// TIA Portal project "Lan-mahai birakaria" (V15.1)

(* hardware
DEVICE "S7-1200 station_1"  S7-1200 Station
   slot 0: "Rack_0"  S7-1200 Rack  Rack  V1.0
   slot 1: "PLC_1"  CPU 1214C AC/DC/Rly  6ES7 214-1BG40-0XB0  V4.0
*)

// ===== PLC "PLC_1"  CPU 1214C AC/DC/Rly =====

VAR_GLOBAL   // PLC tag table "Tabla de variables estándar"
   "Etapa 0" AT %M0.0 : Bool;
   "Etapa 1" AT %M0.1 : Bool;
   "Etapa 2" AT %M0.2 : Bool;
   "Etapa 11" AT %M0.4 : Bool;
   "Etapa 12" AT %M0.5 : Bool;
   "Etapa 20" AT %M0.6 : Bool;
   "Etapa 21" AT %M0.7 : Bool;
   "Etapa 22" AT %M1.0 : Bool;
   "Etapa 23" AT %M1.1 : Bool;
   "Etapa 24" AT %M1.2 : Bool;
   "Etapa 30" AT %M1.3 : Bool;
   "Etapa 31" AT %M1.4 : Bool;
   "Etapa 32" AT %M1.5 : Bool;
   "Etapa 33" AT %M1.6 : Bool;
   "Etapa 34" AT %M1.7 : Bool;
   "Etapa 35" AT %M2.0 : Bool;
   "Etapa 10" AT %M0.3 : Bool;
   "M" AT %I0.0 : Bool;
   "A" AT %I0.1 : Bool;
   "DI0" AT %I0.2 : Bool;
   "DI1" AT %I0.3 : Bool;
   "DI2" AT %I0.4 : Bool;
   "TA" AT %I0.5 : Bool;
   "TB" AT %I0.6 : Bool;
   "TTA" AT %I0.7 : Bool;
   "TTB" AT %I1.0 : Bool;
   "C1R" AT %I1.1 : Bool;
   "C1F" AT %I1.2 : Bool;
   "C2R" AT %I1.3 : Bool;
   "C2F" AT %I1.4 : Bool;
   "S1" AT %Q0.0 : Bool;
   "S2" AT %Q0.1 : Bool;
   "R1" AT %Q0.2 : Bool;
   "R2" AT %Q0.3 : Bool;
   "C1" AT %Q0.4 : Bool;
   "C2" AT %Q0.5 : Bool;
   "MT" AT %Q0.6 : Bool;
   "MP" AT %Q0.7 : Bool;
   "PE" AT %I1.5 : Bool;
END_VAR

// folder: System blocks/Program resources

DATA_BLOCK "Temporizador 1"   // DB1
{ S7_Optimized_Access := 'TRUE' }
AUTHOR : Simatic
FAMILY : IEC
NAME : IEC_TMR
VERSION : 1.0
// stored: InstanceOfName IEC_TIMER
"IEC_TIMER"
BEGIN
END_DATA_BLOCK

DATA_BLOCK "Temporizador 2"   // DB4
{ S7_Optimized_Access := 'TRUE' }
AUTHOR : Simatic
FAMILY : IEC
NAME : IEC_TMR
VERSION : 1.0
// stored: InstanceOfName IEC_TIMER
"IEC_TIMER"
BEGIN
END_DATA_BLOCK

// folder: (top level)

ORGANIZATION_BLOCK "Main"   // OB1, LAD, ProgramCycle
TITLE = "Main Program Sweep (Cycle)"
{ S7_Optimized_Access := 'TRUE' }
VERSION : 0.1
   VAR_INPUT
      Initial_Call : Bool;   // Initial call of this OB
      Remanence : Bool;   // =True, if remanent data are available
   END_VAR
BEGIN

REGION Network 1
   // Etapa 1
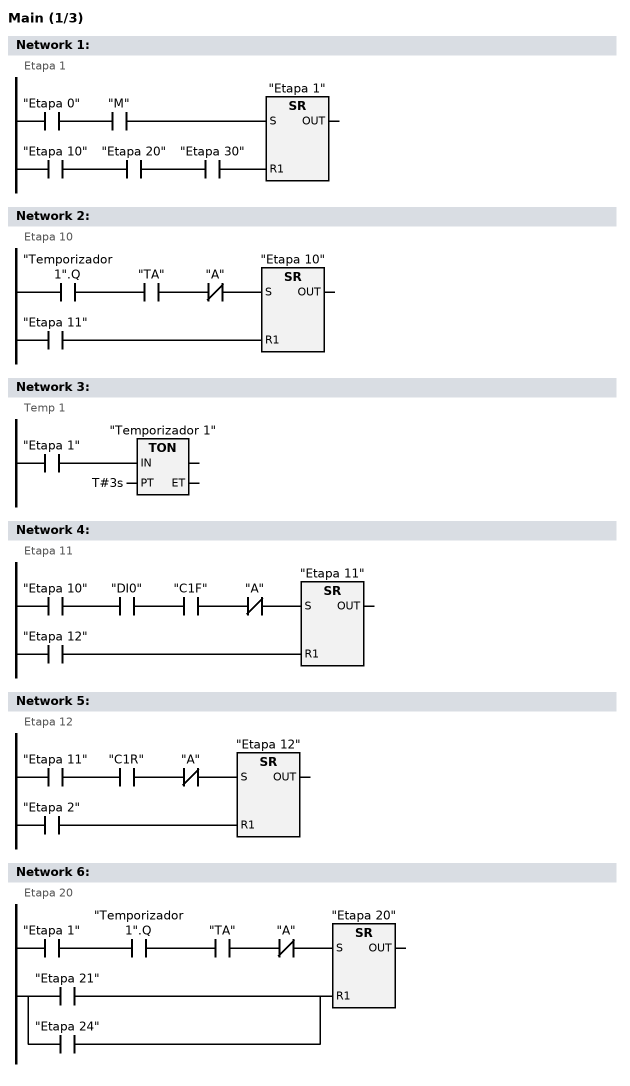
   RUNG wire#powerrail
      Contact( "Etapa 0" )
      Contact( "M" )
      S_SR(operand := "Etapa 1", r1 := wire#w1)
   END_RUNG
   RUNG wire#powerrail
      Contact( "Etapa 10" )
      Contact( "Etapa 20" )
      Contact( "Etapa 30" )
   END_RUNG wire#w1
   // the same network as SCL:
   IF "Etapa 0" AND "M" THEN
       "Etapa 1" := TRUE;   // SR flip-flop
   END_IF;
   IF "Etapa 10" AND "Etapa 20" AND "Etapa 30" THEN "Etapa 1" := FALSE; END_IF;
END_REGION

REGION Network 2
   // Etapa 10
   RUNG wire#powerrail
      Contact( "Temporizador 1".Q )
      Contact( "TA" )
      I_Contact( "A" )
      S_SR(operand := "Etapa 10", r1 := wire#w1)
   END_RUNG
   RUNG wire#powerrail
      Contact( "Etapa 11" )
   END_RUNG wire#w1
   // the same network as SCL:
   IF "Temporizador 1".Q AND "TA" AND NOT "A" THEN
       "Etapa 10" := TRUE;   // SR flip-flop
   END_IF;
   IF "Etapa 11" THEN "Etapa 10" := FALSE; END_IF;
END_REGION

REGION Network 3
   // Temp 1
   "Temporizador 1".TON(IN := "Etapa 1", PT := T#3s);
END_REGION

REGION Network 4
   // Etapa 11
   RUNG wire#powerrail
      Contact( "Etapa 10" )
      Contact( "DI0" )
      Contact( "C1F" )
      I_Contact( "A" )
      S_SR(operand := "Etapa 11", r1 := wire#w1)
   END_RUNG
   RUNG wire#powerrail
      Contact( "Etapa 12" )
   END_RUNG wire#w1
   // the same network as SCL:
   IF "Etapa 10" AND "DI0" AND "C1F" AND NOT "A" THEN
       "Etapa 11" := TRUE;   // SR flip-flop
   END_IF;
   IF "Etapa 12" THEN "Etapa 11" := FALSE; END_IF;
END_REGION

REGION Network 5
   // Etapa 12
   RUNG wire#powerrail
      Contact( "Etapa 11" )
      Contact( "C1R" )
      I_Contact( "A" )
      S_SR(operand := "Etapa 12", r1 := wire#w1)
   END_RUNG
   RUNG wire#powerrail
      Contact( "Etapa 2" )
   END_RUNG wire#w1
   // the same network as SCL:
   IF "Etapa 11" AND "C1R" AND NOT "A" THEN
       "Etapa 12" := TRUE;   // SR flip-flop
   END_IF;
   IF "Etapa 2" THEN "Etapa 12" := FALSE; END_IF;
END_REGION

REGION Network 6
   // Etapa 20
   RUNG wire#powerrail
      Contact( "Etapa 1" )
      Contact( "Temporizador 1".Q )
      Contact( "TA" )
      I_Contact( "A" )
      S_SR(operand := "Etapa 20", r1 := wire#w1)
   END_RUNG
   RUNG wire#powerrail
      Contact( "Etapa 21" )
   END_RUNG wire#w1
   RUNG wire#powerrail
      Contact( "Etapa 24" )
   END_RUNG wire#w1
   // the same network as SCL:
   IF "Etapa 1" AND "Temporizador 1".Q AND "TA" AND NOT "A" THEN
       "Etapa 20" := TRUE;   // SR flip-flop
   END_IF;
   IF "Etapa 21" OR "Etapa 24" THEN "Etapa 20" := FALSE; END_IF;
END_REGION

REGION Network 7
   // Etapa 21
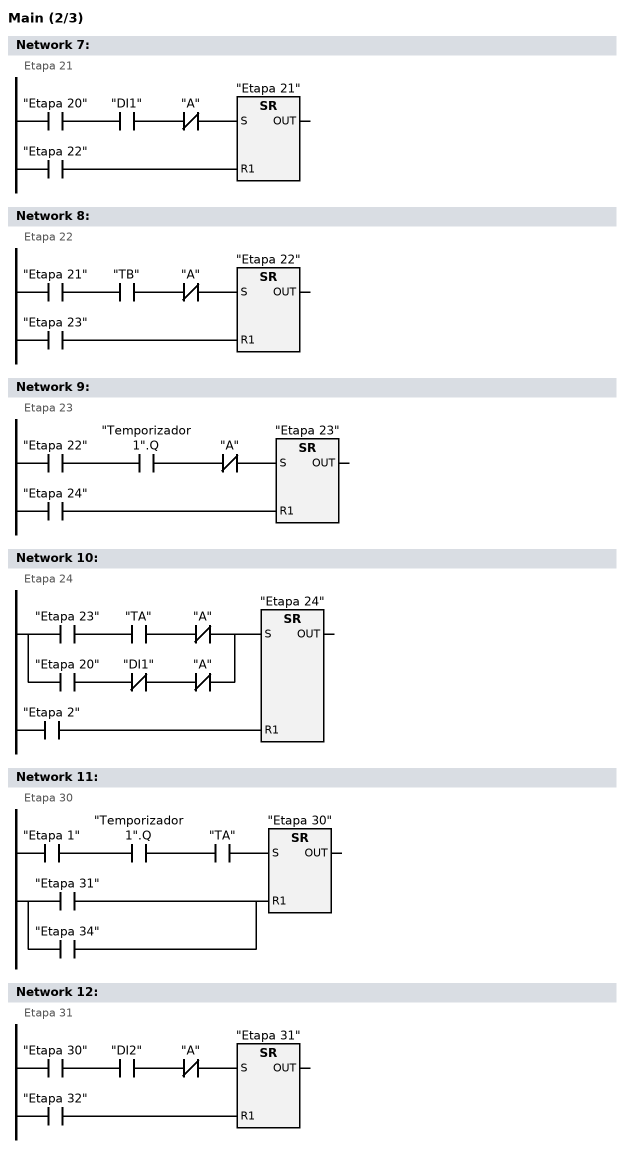
   RUNG wire#powerrail
      Contact( "Etapa 20" )
      Contact( "DI1" )
      I_Contact( "A" )
      S_SR(operand := "Etapa 21", r1 := wire#w1)
   END_RUNG
   RUNG wire#powerrail
      Contact( "Etapa 22" )
   END_RUNG wire#w1
   // the same network as SCL:
   IF "Etapa 20" AND "DI1" AND NOT "A" THEN
       "Etapa 21" := TRUE;   // SR flip-flop
   END_IF;
   IF "Etapa 22" THEN "Etapa 21" := FALSE; END_IF;
END_REGION

REGION Network 8
   // Etapa 22
   RUNG wire#powerrail
      Contact( "Etapa 21" )
      Contact( "TB" )
      I_Contact( "A" )
      S_SR(operand := "Etapa 22", r1 := wire#w1)
   END_RUNG
   RUNG wire#powerrail
      Contact( "Etapa 23" )
   END_RUNG wire#w1
   // the same network as SCL:
   IF "Etapa 21" AND "TB" AND NOT "A" THEN
       "Etapa 22" := TRUE;   // SR flip-flop
   END_IF;
   IF "Etapa 23" THEN "Etapa 22" := FALSE; END_IF;
END_REGION

REGION Network 9
   // Etapa 23
   RUNG wire#powerrail
      Contact( "Etapa 22" )
      Contact( "Temporizador 1".Q )
      I_Contact( "A" )
      S_SR(operand := "Etapa 23", r1 := wire#w1)
   END_RUNG
   RUNG wire#powerrail
      Contact( "Etapa 24" )
   END_RUNG wire#w1
   // the same network as SCL:
   IF "Etapa 22" AND "Temporizador 1".Q AND NOT "A" THEN
       "Etapa 23" := TRUE;   // SR flip-flop
   END_IF;
   IF "Etapa 24" THEN "Etapa 23" := FALSE; END_IF;
END_REGION

REGION Network 10
   // Etapa 24
   RUNG wire#powerrail
      Contact( "Etapa 23" )
      Contact( "TA" )
      I_Contact( "A" )
      wire#w1
      S_SR(operand := "Etapa 24", r1 := wire#w2)
   END_RUNG
   RUNG wire#powerrail
      Contact( "Etapa 20" )
      I_Contact( "DI1" )
      I_Contact( "A" )
   END_RUNG wire#w1
   RUNG wire#powerrail
      Contact( "Etapa 2" )
   END_RUNG wire#w2
   // the same network as SCL:
   IF ("Etapa 23" AND "TA" AND NOT "A") OR ("Etapa 20" AND NOT "DI1" AND NOT "A") THEN
       "Etapa 24" := TRUE;   // SR flip-flop
   END_IF;
   IF "Etapa 2" THEN "Etapa 24" := FALSE; END_IF;
END_REGION

REGION Network 11
   // Etapa 30
   RUNG wire#powerrail
      Contact( "Etapa 1" )
      Contact( "Temporizador 1".Q )
      Contact( "TA" )
      S_SR(operand := "Etapa 30", r1 := wire#w1)
   END_RUNG
   RUNG wire#powerrail
      Contact( "Etapa 31" )
   END_RUNG wire#w1
   RUNG wire#powerrail
      Contact( "Etapa 34" )
   END_RUNG wire#w1
   // the same network as SCL:
   IF "Etapa 1" AND "Temporizador 1".Q AND "TA" THEN
       "Etapa 30" := TRUE;   // SR flip-flop
   END_IF;
   IF "Etapa 31" OR "Etapa 34" THEN "Etapa 30" := FALSE; END_IF;
END_REGION

REGION Network 12
   // Etapa 31
   RUNG wire#powerrail
      Contact( "Etapa 30" )
      Contact( "DI2" )
      I_Contact( "A" )
      S_SR(operand := "Etapa 31", r1 := wire#w1)
   END_RUNG
   RUNG wire#powerrail
      Contact( "Etapa 32" )
   END_RUNG wire#w1
   // the same network as SCL:
   IF "Etapa 30" AND "DI2" AND NOT "A" THEN
       "Etapa 31" := TRUE;   // SR flip-flop
   END_IF;
   IF "Etapa 32" THEN "Etapa 31" := FALSE; END_IF;
END_REGION

REGION Network 13
   // Etapa 32
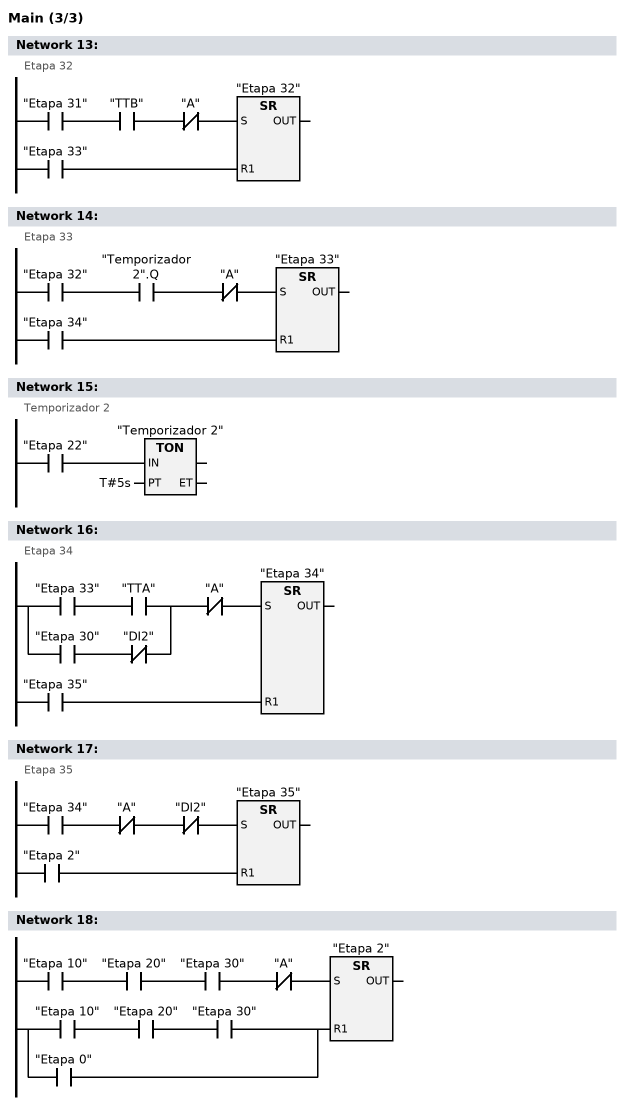
   RUNG wire#powerrail
      Contact( "Etapa 31" )
      Contact( "TTB" )
      I_Contact( "A" )
      S_SR(operand := "Etapa 32", r1 := wire#w1)
   END_RUNG
   RUNG wire#powerrail
      Contact( "Etapa 33" )
   END_RUNG wire#w1
   // the same network as SCL:
   IF "Etapa 31" AND "TTB" AND NOT "A" THEN
       "Etapa 32" := TRUE;   // SR flip-flop
   END_IF;
   IF "Etapa 33" THEN "Etapa 32" := FALSE; END_IF;
END_REGION

REGION Network 14
   // Etapa 33
   RUNG wire#powerrail
      Contact( "Etapa 32" )
      Contact( "Temporizador 2".Q )
      I_Contact( "A" )
      S_SR(operand := "Etapa 33", r1 := wire#w1)
   END_RUNG
   RUNG wire#powerrail
      Contact( "Etapa 34" )
   END_RUNG wire#w1
   // the same network as SCL:
   IF "Etapa 32" AND "Temporizador 2".Q AND NOT "A" THEN
       "Etapa 33" := TRUE;   // SR flip-flop
   END_IF;
   IF "Etapa 34" THEN "Etapa 33" := FALSE; END_IF;
END_REGION

REGION Network 15
   // Temporizador 2
   "Temporizador 2".TON(IN := "Etapa 22", PT := T#5s);
END_REGION

REGION Network 16
   // Etapa 34
   RUNG wire#powerrail
      Contact( "Etapa 33" )
      Contact( "TTA" )
      wire#w1
      I_Contact( "A" )
      S_SR(operand := "Etapa 34", r1 := wire#w2)
   END_RUNG
   RUNG wire#powerrail
      Contact( "Etapa 30" )
      I_Contact( "DI2" )
   END_RUNG wire#w1
   RUNG wire#powerrail
      Contact( "Etapa 35" )
   END_RUNG wire#w2
   // the same network as SCL:
   IF (("Etapa 33" AND "TTA") OR ("Etapa 30" AND NOT "DI2")) AND NOT "A" THEN
       "Etapa 34" := TRUE;   // SR flip-flop
   END_IF;
   IF "Etapa 35" THEN "Etapa 34" := FALSE; END_IF;
END_REGION

REGION Network 17
   // Etapa 35
   RUNG wire#powerrail
      Contact( "Etapa 34" )
      I_Contact( "A" )
      I_Contact( "DI2" )
      S_SR(operand := "Etapa 35", r1 := wire#w1)
   END_RUNG
   RUNG wire#powerrail
      Contact( "Etapa 2" )
   END_RUNG wire#w1
   // the same network as SCL:
   IF "Etapa 34" AND NOT "A" AND NOT "DI2" THEN
       "Etapa 35" := TRUE;   // SR flip-flop
   END_IF;
   IF "Etapa 2" THEN "Etapa 35" := FALSE; END_IF;
END_REGION

REGION Network 18
   RUNG wire#powerrail
      Contact( "Etapa 10" )
      Contact( "Etapa 20" )
      Contact( "Etapa 30" )
      I_Contact( "A" )
      S_SR(operand := "Etapa 2", r1 := wire#w1)
   END_RUNG
   RUNG wire#powerrail
      Contact( "Etapa 10" )
      Contact( "Etapa 20" )
      Contact( "Etapa 30" )
   END_RUNG wire#w1
   RUNG wire#powerrail
      Contact( "Etapa 0" )
   END_RUNG wire#w1
   // the same network as SCL:
   IF "Etapa 10" AND "Etapa 20" AND "Etapa 30" AND NOT "A" THEN
       "Etapa 2" := TRUE;   // SR flip-flop
   END_IF;
   IF ("Etapa 10" AND "Etapa 20" AND "Etapa 30") OR "Etapa 0" THEN "Etapa 2" := FALSE; END_IF;
END_REGION
END_ORGANIZATION_BLOCK

ORGANIZATION_BLOCK "Startup"   // OB100, LAD, Startup
TITLE = "Complete Restart"
{ S7_Optimized_Access := 'TRUE' }
VERSION : 0.1
   VAR_INPUT
      LostRetentive : Bool;   // True if retentive data are lost
      LostRTC : Bool;   // True if date and time are lost
   END_VAR
BEGIN

REGION Network 1
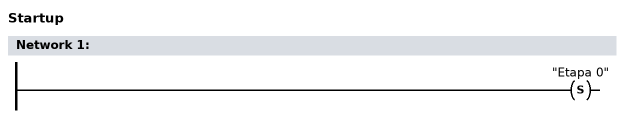
   RUNG wire#powerrail
      S_Coil( "Etapa 0" )
   END_RUNG
   // the same network as SCL:
   "Etapa 0" := TRUE;
END_REGION
END_ORGANIZATION_BLOCK